{attribute addProperty BoxType "EL5101-0010-0019"}
{attribute addProperty Id "ENC_Status_compactAT %I*ENC_Status_compact_6BB1ED4B4860ENC_Control_compactAT %Q*ENC_Control_compact_03701F333240WcStateAT %I*WcState_98A4DF7520.250InfoDataAT %I*InfoData_BC63D37F80100"}
{attribute addProperty CRC "4280390666"}
{attribute addProperty SizeInBites "162"}
{attribute addProperty SizeInBytes "20.25"}
TYPE EL5101_354B2489 :
STRUCT
	{attribute addProperty Name "ENC_Status_compact"}
	ENC_Status_compact : ENC_Status_compact_6BB1ED4B;
	{attribute addProperty Name "ENC_Control_compact"}
	ENC_Control_compact : ENC_Control_compact_03701F33;
	{attribute addProperty Name "WcState"}
	WcState : WcState_98A4DF75;
	{attribute addProperty Name "InfoData"}
	InfoData : InfoData_BC63D37F;
END_STRUCT
END_TYPE

(* stored: Version 1.2.0.0, ProductVersion 3.1.4024.9
   DUT EL5101_354B2489: Id {1bf307f0-781e-4785-a55a-2c5d1b1898c3} *)
